FUNCTION_BLOCK MainAxisRot
VAR_INPUT
	Input1:BOOL;
	InputTargetSpeed	:	REAL;
	ForwardRotFlag	:	BOOL;
	BackwardRotFlag	:	BOOL;
END_VAR
VAR_OUTPUT
END_VAR
VAR
	temp1, temp2 	:	MC_MoveVelocity;
	AxisStop	:	MC_Stop;
	trig1, trig2	: 	F_TRIG;
END_VAR
VAR // added by the converter: edge detectors and wires of the graphical bodies
    _w1, _w2 : ANY;
END_VAR

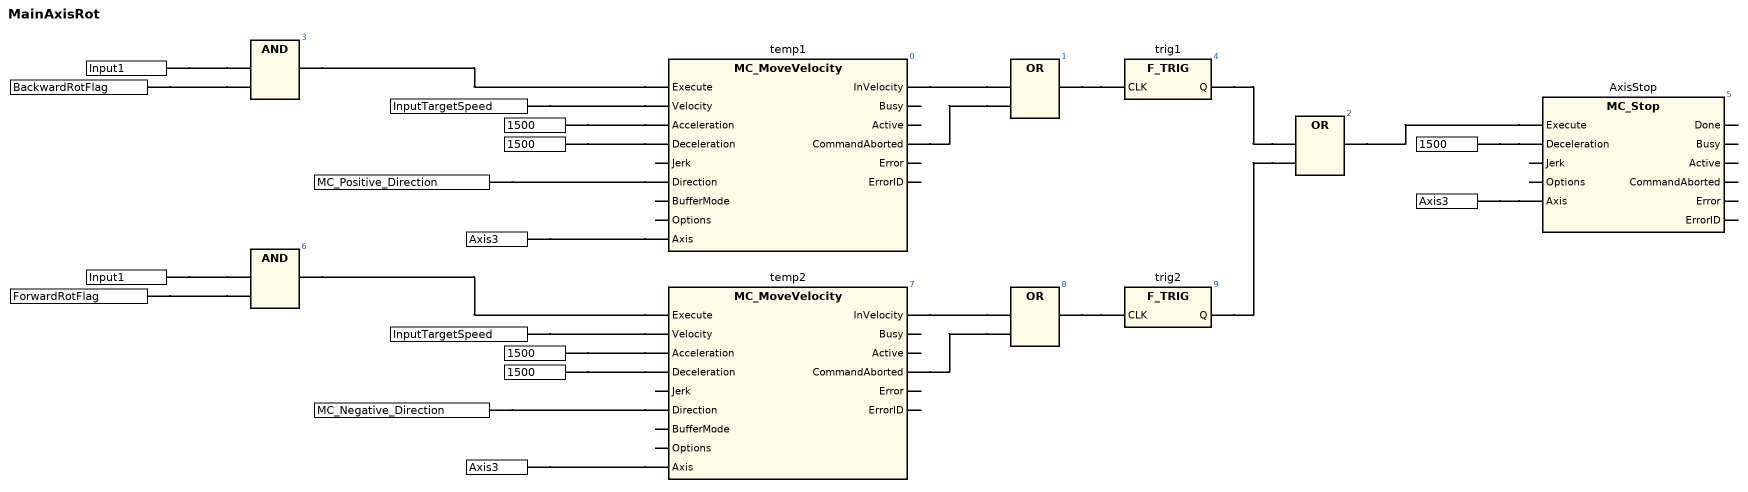
temp1(
    Execute := _w1,
    Velocity := InputTargetSpeed,
    Acceleration := 1500,
    Deceleration := 1500,
    Direction := MC_Positive_Direction,
    Axis := Axis3); // MC_MoveVelocity
_w2 := trig1.Q OR trig2.Q;
_w1 := Input1 AND BackwardRotFlag;
trig1(CLK := temp1.InVelocity OR temp1.CommandAborted); // F_TRIG
AxisStop(Execute := _w2, Deceleration := 1500, Axis := Axis3); // MC_Stop
temp2(
    Execute := Input1 AND ForwardRotFlag,
    Velocity := InputTargetSpeed,
    Acceleration := 1500,
    Deceleration := 1500,
    Direction := MC_Negative_Direction,
    Axis := Axis3); // MC_MoveVelocity
trig2(CLK := temp2.InVelocity OR temp2.CommandAborted); // F_TRIG

END_FUNCTION_BLOCK

(* stored: Version 1.1.0.1, ProductVersion 3.1.4024.12
   POU MainAxisRot: Id {eecbddfd-4f72-4a79-b0e3-44240909a517}, SpecialFunc None *)
